Fanuc KAREL source: kt00442.compact.KL

PROGRAM KT00442
%STACKSIZE=65535
%PRIORITY=65535
%NOLOCKGROUP
VAR
R1 : REAL
R2 : REAL
OUT : BOOLEAN
BEGIN
R1=2.0
R2=3.0
R1=2.0
R2=3.0
OUT=(R1 >=R2)
END KT00442
